# B&R Automation Studio project Parker_BMM_ST_V5_3147_V12 (part 2)

### Acp10map.ncm - 5PPC2100_BY01_000/Motion/Acp10map.ncm
```
NcMapping (NcSwId=Acp10, DisabledNodesAreHidden=True)
  NcObject 8V1090.001-2_ncV_AXIS1 (ModuleId=8V1090.001-2_L_BlowPin, Type=ncV_AXIS, Channel=1, Disabled=TRUE, ModuleDisabled=FALSE)
  NcObject 8V1090.001-2a_ncV_AXIS1 (ModuleId=8V1090.001-2a_R_BlowPin, Type=ncV_AXIS, Channel=1, Disabled=TRUE, ModuleDisabled=FALSE)
  NcObject 8V1180.001-2_ncV_AXIS1 (ModuleId=8V1180.001-2_L_Carriage, Type=ncV_AXIS, Channel=1, Disabled=TRUE, ModuleDisabled=FALSE)
  NcObject 8V1180.001-2a_ncV_AXIS1 (ModuleId=8V1180.001-2a_R_Carriage, Type=ncV_AXIS, Channel=1, Disabled=TRUE, ModuleDisabled=FALSE)
  NcObject 8B0P0440HW00.001-1_ncAXIS2 (ModuleId=8B0P0440HW00.001-1, Type=ncAXIS, Channel=2, AcoposSimulation=Off, Disabled=TRUE, ModuleDisabled=FALSE)
  NcObject 8B0P0440HW00.001-1_ncV_AXIS1 (ModuleId=8B0P0440HW00.001-1, Type=ncV_AXIS, Channel=1, Disabled=TRUE, ModuleDisabled=FALSE)
  NcObject 8B0P0440HW00.001-1_ncV_AXIS2 (ModuleId=8B0P0440HW00.001-1, Type=ncV_AXIS, Channel=2, Disabled=TRUE, ModuleDisabled=FALSE)
  NcObject 8BVI0110HWS0.000-1_ncAXIS2 (ModuleId=8BVI0110HWS0.000-1, Type=ncAXIS, Channel=2, AcoposSimulation=Off, Disabled=TRUE, ModuleDisabled=FALSE)
  NcObject 8BVI0110HWS0.000-1_ncV_AXIS1 (ModuleId=8BVI0110HWS0.000-1, Type=ncV_AXIS, Channel=1, Disabled=TRUE, ModuleDisabled=FALSE)
  NcObject 8BVI0110HWS0.000-1_ncV_AXIS2 (ModuleId=8BVI0110HWS0.000-1, Type=ncV_AXIS, Channel=2, Disabled=TRUE, ModuleDisabled=FALSE)
  NcObject gAxisBlowPinL (ModuleId=8V1090.001-2_L_BlowPin, Type=ncAXIS, Channel=1, AcoposSimulation=Off, InitParameter=BlowPinL, AcoposParameter=BlowPinLR, Disabled=TRUE, ModuleDisabled=FALSE)
  NcObject gAxisBlowPinR (ModuleId=8V1090.001-2a_R_BlowPin, Type=ncAXIS, Channel=1, AcoposSimulation=Off, InitParameter=BlowPinR, AcoposParameter=BlowPinLR, Disabled=TRUE, ModuleDisabled=FALSE)
  NcObject gAxisCarriageL (ModuleId=8V1180.001-2_L_Carriage, Type=ncAXIS, Channel=1, AcoposSimulation=Off, InitParameter=CarriageL, AcoposParameter=CarraigeLR, Disabled=TRUE, ModuleDisabled=FALSE)
  NcObject gAxisCarriageR (ModuleId=8V1180.001-2a_R_Carriage, Type=ncAXIS, Channel=1, AcoposSimulation=Off, InitParameter=CarriageR, AcoposParameter=CarraigeLR, Disabled=TRUE, ModuleDisabled=FALSE)
  NcObject 8BVI0330HWS0.000-1_ncAXIS2 (ModuleId=8BVI0330HWS0.000-1, Type=ncAXIS, Channel=2, AcoposSimulation=Off, Disabled=TRUE, ModuleDisabled=FALSE)
  NcObject 8BVI0330HWS0.000-1_ncV_AXIS1 (ModuleId=8BVI0330HWS0.000-1, Type=ncV_AXIS, Channel=1, Disabled=TRUE, ModuleDisabled=FALSE)
  NcObject 8BVI0330HWS0.000-1_ncV_AXIS2 (ModuleId=8BVI0330HWS0.000-1, Type=ncV_AXIS, Channel=2, Disabled=TRUE, ModuleDisabled=FALSE)
  NcObject 8BVI0330HWS0.000-1a_ncAXIS2 (ModuleId=8BVI0330HWS0.000-1a, Type=ncAXIS, Channel=2, AcoposSimulation=Off, Disabled=TRUE, ModuleDisabled=FALSE)
  NcObject 8BVI0330HWS0.000-1a_ncV_AXIS1 (ModuleId=8BVI0330HWS0.000-1a, Type=ncV_AXIS, Channel=1, Disabled=TRUE, ModuleDisabled=FALSE)
  NcObject 8BVI0330HWS0.000-1a_ncV_AXIS2 (ModuleId=8BVI0330HWS0.000-1a, Type=ncV_AXIS, Channel=2, Disabled=TRUE, ModuleDisabled=FALSE)
  NcObject 8BVI0110HWD0.000-1_ncV_AXIS1 (ModuleId=8BVI0110HWD0.000-1, Type=ncV_AXIS, Channel=1, Disabled=TRUE, ModuleDisabled=FALSE)
  NcObject 8BVI0110HWD0.000-1_ncV_AXIS2 (ModuleId=8BVI0110HWD0.000-1, Type=ncV_AXIS, Channel=2, Disabled=TRUE, ModuleDisabled=FALSE)
  NcObject 8BVI0440HWS0.000-1a_ncAXIS2 (ModuleId=8BVI0440HWS0.000-1a, Type=ncAXIS, Channel=2, AcoposSimulation=Off, Disabled=TRUE, ModuleDisabled=FALSE)
  NcObject 8BVI0440HWS0.000-1a_ncV_AXIS1 (ModuleId=8BVI0440HWS0.000-1a, Type=ncV_AXIS, Channel=1, Disabled=TRUE, ModuleDisabled=FALSE)
  NcObject 8BVI0440HWS0.000-1a_ncV_AXIS2 (ModuleId=8BVI0440HWS0.000-1a, Type=ncV_AXIS, Channel=2, Disabled=TRUE, ModuleDisabled=FALSE)
  NcObject 8BVI0028HWD0.000-1_ncV_AXIS1 (ModuleId=8BVI0028HWD0.000-1, Type=ncV_AXIS, Channel=1, Disabled=TRUE, ModuleDisabled=FALSE)
  NcObject 8BVI0028HWD0.000-1_ncV_AXIS2 (ModuleId=8BVI0028HWD0.000-1, Type=ncV_AXIS, Channel=2, Disabled=TRUE, ModuleDisabled=FALSE)
  NcObject gAxisTransferR (ModuleId=8BVI0110HWS0.000-1, Type=ncAXIS, Channel=1, AcoposSimulation=Off, InitParameter=TransferR, AcoposParameter=Tansfer, Disabled=TRUE, ModuleDisabled=FALSE)
  NcObject gAxisTransferR (ModuleId=8BVI0110HWS0.000-1, Type=ncAXIS, Channel=1, AcoposSimulation=Off, InitParameter=TransferR, AcoposParameter=Tansfer, Disabled=TRUE, ModuleDisabled=FALSE)
  NcObject gAxisCarriageL (ModuleId=8BVI0330HWS0.000-1a, Type=ncAXIS, Channel=1, AcoposSimulation=Off, InitParameter=CarriageL, AcoposParameter=CarraigeLR, Disabled=TRUE, ModuleDisabled=FALSE)
  NcObject 8BVI0330HWS0.000-1b_ncAXIS2 (ModuleId=8BVI0330HWS0.000-1b, Type=ncAXIS, Channel=2, AcoposSimulation=Off, Disabled=TRUE, ModuleDisabled=FALSE)
  NcObject 8BVI0330HWS0.000-1b_ncV_AXIS1 (ModuleId=8BVI0330HWS0.000-1b, Type=ncV_AXIS, Channel=1, Disabled=TRUE, ModuleDisabled=FALSE)
  NcObject 8BVI0330HWS0.000-1b_ncV_AXIS2 (ModuleId=8BVI0330HWS0.000-1b, Type=ncV_AXIS, Channel=2, Disabled=TRUE, ModuleDisabled=FALSE)
  NcObject 8BVI0440HWS0.000-1_ncAXIS2 (ModuleId=8BVI0440HWS0.000-1, Type=ncAXIS, Channel=2, AcoposSimulation=Off, Disabled=TRUE, ModuleDisabled=FALSE)
  NcObject 8BVI0440HWS0.000-1_ncV_AXIS1 (ModuleId=8BVI0440HWS0.000-1, Type=ncV_AXIS, Channel=1, Disabled=TRUE, ModuleDisabled=FALSE)
  NcObject 8BVI0440HWS0.000-1_ncV_AXIS2 (ModuleId=8BVI0440HWS0.000-1, Type=ncV_AXIS, Channel=2, Disabled=TRUE, ModuleDisabled=FALSE)
  NcObject gAxisClampR (ModuleId=8BVI0440HWS0.000-1, Type=ncAXIS, Channel=1, AcoposSimulation=Off, InitParameter=ClampR, AcoposParameter=ClampLR, Disabled=FALSE, ModuleDisabled=FALSE)
  NcObject gAxisClampR (ModuleId=8BVI0330HWS0.000-1b, Type=ncAXIS, Channel=1, AcoposSimulation=Off, InitParameter=ClampR, AcoposParameter=ClampLR, Disabled=TRUE, ModuleDisabled=FALSE)
  NcObject gAxisClampL (ModuleId=8BVI0440HWS0.000-1a, Type=ncAXIS, Channel=1, AcoposSimulation=Off, InitParameter=ClampL, AcoposParameter=ClampLR, Disabled=TRUE, ModuleDisabled=FALSE)
  NcObject gAxisExtrlift (ModuleId=8BVI0028HWD0.000-1, Type=ncAXIS, Channel=1, AcoposSimulation=Off, InitParameter=ExtrLift1, AcoposParameter=ExtrLift2, Disabled=FALSE, ModuleDisabled=FALSE)
  NcObject gAxisTransferR (ModuleId=8BVI0028HWD0.000-1, Type=ncAXIS, Channel=2, AcoposSimulation=Off, InitParameter=TransferR, AcoposParameter=Tansfer, Disabled=FALSE, ModuleDisabled=FALSE)
  NcObject gAxisPwr (ModuleId=8B0P0440HW00.001-1, Type=ncAXIS, Channel=1, AcoposSimulation=Off, InitParameter=Power, AcoposParameter=Power1, Disabled=FALSE, ModuleDisabled=FALSE)
  NcObject gAxisCarriageR (ModuleId=8BVI0330HWS0.000-1, Type=ncAXIS, Channel=1, AcoposSimulation=Off, InitParameter=CarriageR, AcoposParameter=CarraigeLR, Disabled=FALSE, ModuleDisabled=FALSE)
  NcObject gAxisThick (ModuleId=8BVI0110HWD0.000-1, Type=ncAXIS, Channel=1, AcoposSimulation=Off, InitParameter=ThickInit, AcoposParameter=ThickPara, Disabled=FALSE, ModuleDisabled=FALSE)
  NcObject gAxisBlowPinR (ModuleId=8BVI0110HWD0.000-1, Type=ncAXIS, Channel=2, AcoposSimulation=Off, InitParameter=BlowPinR, AcoposParameter=BlowPinLR, Disabled=FALSE, ModuleDisabled=FALSE)
```

## Configuration AR000

CPU PC_any, AutomationRuntime D4.26, Build 4.1.2, Vc V4.26.8, Safety 0.0

### Task classes (Cpu.sw)
```
Cyclic#1 (cycle 2000 us, tolerance 0 us):
  tk1_in <- In_Out.tk1_in.prg
  timer <- process.timer.prg
  length <- process.length.prg
  clamp <- process.clamp.prg
  carriage <- process.carriage.prg
  blowpin <- process.blowpin.prg
  tk1_out <- In_Out.tk1_out.prg
Cyclic#2 (cycle 10000 us, tolerance 100000 us):
  h_pwm <- Heating.h_pwm.prg
  tk2_io <- In_Out.tk2_io.prg
Cyclic#3 (cycle 4000 us, tolerance 100000 us):
  extrlift <- process.extrlift.prg
  cutter <- process.cutter.prg
  cutneck <- process.cutneck.prg
  cooldef <- process.cooldef.prg
  blowdef <- process.blowdef.prg
  bdeflash <- process.bdeflash.prg
  tdeflash <- process.tdeflash.prg
  inerpin <- process.inerpin.prg
  highblow <- process.highblow.prg
  lowblow <- process.lowblow.prg
  coolpin <- process.coolpin.prg
  coolpin2 <- process.coolpin2.prg
  coolpin3 <- process.coolpin3.prg
  submold <- process.submold.prg
  pinpart <- process.pinpart.prg
  screw <- process.screw.prg
  sealer <- process.sealer.prg
  bblowpin <- process.bblowpin.prg
  support <- process.support.prg
  tonnage <- process.tonnage.prg
  robot <- process.robot.prg
  extruder <- machine.extruder.prg
  extru_plk <- machine.extru_plk.prg
  autorun <- process.autorun.prg
Cyclic#4 (cycle 20000 us, tolerance 200000 us):
  keyled <- screen.keyled.prg
  manual <- machine.manual.prg
  calib <- machine.calib.prg
  reset <- machine.reset.prg
  workmode <- machine.workmode.prg
  mode <- machine.mode.prg
  panel <- screen.panel.prg
  hmi_cpy <- screen.hmi_cpy.prg
  pump <- machine.pump.prg
  mac_lubr <- machine.mac_lubr.prg
  oil_accu <- machine.oil_accu.prg
  mbusMaster <- comm.mbusMaster.prg
Cyclic#5 (cycle 500000 us, tolerance 500000 us):
  h_pid <- Heating.h_pid.prg
Cyclic#8 (cycle 200000 us, tolerance 30000000 us):
  spc_ctrl <- spc.spc_ctrl.prg
  trend <- Heating.trend.prg
  h_plan <- Heating.h_plan.prg
  scrshot <- screen.scrshot.prg
  hmiset <- screen.hmiset.prg
  password <- screen.password.prg
  modem <- comm.modem.prg
  vpn <- screen.vpn.prg
  recipe <- recipeMan.recipe.prg
  multsave <- recipeMan.multsave.prg
  oncesave <- recipeMan.oncesave.prg
  cfg_cpy <- recipeMan.cfg_cpy.prg
  pvchg <- VarChgLog.pvchg.prg
  alarm <- machine.alarm.prg
  epl <- comm.epl.prg
  energy <- machine.energy.prg
DataObjects: mb_cmd <- comm.mb_cmd.dob, pv_chg <- VarChgLog.pv_chg.dob, var_fix <- recipeMan.var_fix.dob, var_mold <- recipeMan.var_mold.dob, cfg_dat <- recipeMan.cfg_dat.dob, Acp10sys
VcDataObjects: visu15 <- Visu.visu15.dob
Binaries: TCData, visu1502, vccnum, vcpdvnc, vccalarm, vccovl, vcshared, vcfile, vccstr, vccline, arial, vcctrend, vcchtml, vcgclass, tahomabd, vccbtn, vcrt, vccdbox, visu1503, vcclbox, simsun, vcctext, vccbmp, vcfntttf, vcalarm, vcdsint, vcnet, visu1501, vccshape, vcchspot, arialbd, vctcal, vcmgr, vcdsloc, myxh, visvc, tahoma, vccurl, vccdt, vccbar, vcpfar00, vcpdsw, vcxml, vccscale, vcbclass, iomap, sysconf, ashwd, asfw, User, arconfig, Role, Acp10map, acp10cfg
Libraries: visapi, FileIO, runtime, sys_lib, standard, operator, dvframe, DataObj, Convert, brsystem, astime, asstring, AsIO, AsArLog, AsARCfg, Motorky, DRV_mbus, LoopConR, SimpFun, HydCtrl, NcGlobal, Acp10par, Acp10_MC, AsEPL, powerlnk, vcresman, ashydcon
```

### Hardware
```
PC : PC_any v1.1.0.0 (OrderNumber=PC)
  Connector IF3:
    Vnc1
    VncVcObjectName1 = visu15
    VncAuthentication1 = 1
    VncPasswordViewOnly1 = 1
    VncPasswordViewControl1 = 2
  ConfigurationID = bmm_AR000
  PermanentPvSize = 10000
  RemanentGlobalPvSize = 20000
  SystemTick = 2000
  TaskClassIdleTime = 2000
  Cyclic1Duration = 2000
  Cyclic1Tolerance = 0
  Cyclic1Output = 1
  Cyclic2Duration = 10000
  Cyclic2Tolerance = 100000
  Cyclic3Duration = 4000
  Cyclic3Tolerance = 100000
  Cyclic4Duration = 20000
  Cyclic4Tolerance = 200000
  Cyclic5Duration = 500000
  Cyclic5Tolerance = 500000
  Cyclic5Stack = 20000
  Cyclic6Duration = 30000
  Cyclic6Tolerance = 3000000
  Cyclic7Duration = 90000
  Cyclic7Tolerance = 9000000
  Cyclic8Duration = 200000
  Cyclic8Tolerance = 30000000
  Cyclic8Stack = 30000
```

### Acp10cfg.ncc - PC/Motion/Acp10cfg.ncc
```
NcConfiguration (Version=2.52.5, NcSwId=Acp10)
  ACP10CF1_typ:
    cnt_nettrc_rec_drive = 150
    bufsize_trace_upload = 1200
    tc_nc_man_task = Cyclic #1
    glob_pv_as_ncobject = Yes
    ncsys_dl_broadcast = Yes
    ncsys_dl_acp_reset = Yes
    safemc_log_err_to_ax = Yes
    network_init:
      ncsw_init_execute = Yes
      automatic_execute = No
      node_nr_warning = Yes
      net_err_before_ncact = Yes
    nettrc:
      enter_parsecrec = Yes
      enter_ncaction = Yes
      save_ring_startidx = No
    cam_prof_download:
      cam_dat_dl_parallel = No
      tc_cam_dl_parallel = Task class for NC Manager task
```

## Logical view

Binary libraries used (declarations not repeated): visapi, FileIO, runtime, sys_lib, standard, operator, dvframe, DataObj, Convert, brsystem, astime, asstring, AsIO, AsArLog, AsARCfg, Motorky 2.16.0, DRV_mbus, LoopConR 2.80.2, vcscrsht 4.24.0, HydCtrl 1.03.0, AsHydCon 3.10.0, AsEPL, Acp10man 5.06.1, Acp10par 5.06.1, NcGlobal 5.06.1, Acp10sim 5.06.1, Acp10_MC 5.06.1

### Package Logical/GlobalIncludes - Global include file

### draw.h
```c
#ifndef draw_h_
#define draw_h_

#define VSCREEN_WIDTH               302
#define VSCREEN_HEIGHT              402
#define VSCREEN_X0_POSITION         150
#define VSCREEN_Y0_POSITION          85

#define VSCREEN_COLOR_WEIGHT        169
#define VSCREEN_COLOR_BACKGROUND    140
#define VSCREEN_COLOR_FOCUS_LINE  	 51
#define VSCREEN_COLOR_UNFOCUS_LINE 	200
#define VSCREEN_COLOR_CURVE  	       46

#define VSCREEN_COLOR_CROSS_CURSOR 	 44
#define VSCREEN_COLOR_FRAME      	  0

#define S$THICK_POINT		   400
#define S$THICK_X_LENGTH		3000

#define S$THICK_INIT_LENGTH   300

#define S$THICK_SAMPLE		   100
#define S$THICK_MAX		      399
#define S$THICK_V_SCALE		   4

#define S$STEP_EDIT			10
#define S$STEP_ADDLINE     20
#define S$STEP_DELLINE	   30
#define S$STEP_CURVETOL		40
#define S$STEP_CURVEMOVE	50
#define S$STEP_UNDO			60
#define S$STEP_REDO			65
#define S$STEP_CLAER			70

#endif
```

### keyap880.h
```c
#ifndef keyap880_h_
#define keyap880_h_

#define S$KEYMATRIX_MAXCOUNT    400

#define OFFSET_EX2_01            216

/*  0 -- 39 AP880 key */
#define S$KEYMATRIX_MAIN_PUMP   	   0
#define S$KEYMATRIX_PARISON_PUMP 	1
#define S$KEYMATRIX_EXTRUDER_A   	2
#define S$KEYMATRIX_EXTRUDER_B   	3

#define S$KEYMATRIX_MODE_CALIB   	4
#define S$KEYMATRIX_MODE_MANUAL  	5
#define S$KEYMATRIX_MODE_AUTO    	6
#define S$KEYMATRIX_AUTO_RESET   	7
#define S$KEYMATRIX_CUTTER_FW   		8
#define S$KEYMATRIX_EXTRUDER_UP  	9
#define S$KEYMATRIX_LUBRICATION     10
#define S$KEYMATRIX_ALARM_RESET     11

#define S$KEYMATRIX_F1   				12
#define S$KEYMATRIX_F2   				13
#define S$KEYMATRIX_F3   				14
#define S$KEYMATRIX_F4   				15
#define S$KEYMATRIX_F5   				16
#define S$KEYMATRIX_F6   				17
#define S$KEYMATRIX_F7   				18
#define S$KEYMATRIX_F8   				19
#define S$KEYMATRIX_F9   				20
#define S$KEYMATRIX_F10   				21
#define S$KEYMATRIX_F11   				22
#define S$KEYMATRIX_F12   				23
#define S$KEYMATRIX_F13   				24
#define S$KEYMATRIX_F14   				25
#define S$KEYMATRIX_F15   				26
#define S$KEYMATRIX_F16   				27

#define S$KEYMATRIX_CARRIAGE_UP  	28
#define S$KEYMATRIX_CARRIAGE_DN  	29
#define S$KEYMATRIX_CLAMP_OPN   		30
#define S$KEYMATRIX_CLAMP_CLS   		31
#define S$KEYMATRIX_BLOWPIN_UP   	32
#define S$KEYMATRIX_BLOWPIN_DN   	33
#define S$KEYMATRIX_TOP_DEFLASH_FW  34
#define S$KEYMATRIX_BOT_DEFLASH_FW  35
#define S$KEYMATRIX_ROBOT_FW   		36
#define S$KEYMATRIX_ROBOT_BW   		37
#define S$KEYMATRIX_ROBOT_DN   		38
#define S$KEYMATRIX_ROBOT_CLS 		39

/*   5AC800EXT2-01 key   offset 216 */
#define S$KEYMATRIX_NUM7   		 	60
#define S$KEYMATRIX_NUM8   		 	61
#define S$KEYMATRIX_NUM9   		 	62
#define S$KEYMATRIX_NUM4   		 	64
#define S$KEYMATRIX_NUM5   		 	65
#define S$KEYMATRIX_NUM6   		 	66
#define S$KEYMATRIX_NUM1   		 	68
#define S$KEYMATRIX_NUM2   			69
#define S$KEYMATRIX_NUM3   		 	70
#define S$KEYMATRIX_NUM0   		 	73

#define S$KEYMATRIX_ESC    		 	63
#define S$KEYMATRIX_DEL			 		67
#define S$KEYMATRIX_ENTER  	     	71
#define S$KEYMATRIX_TAB          	77
#define S$KEYMATRIX_UP					75
#define S$KEYMATRIX_DOWN				79
#define S$KEYMATRIX_LEFT				76
#define S$KEYMATRIX_RIGHT				78

/* reserve key  */
#define S$KEYMATRIX_TOP_DEFLASH_BW  101
#define S$KEYMATRIX_ROBOT_UP   		102

#define S$KEYMATRIX_ROBOT_REJECT    103
#define S$KEYMATRIX_ROBOT_RESET 		104
#define S$KEYMATRIX_SUPPORT   		105
#define S$KEYMATRIX_SPEED_UP   		106
#define S$KEYMATRIX_SPEED_DN   	   107
#define S$KEYMATRIX_COOL_DEFLASH    108
#define S$KEYMATRIX_BLOW         	109
#define S$KEYMATRIX_BLOW_LOW        110
#define S$KEYMATRIX_COOL_DN         111
#define S$KEYMATRIX_COOL_BLOW			112
#define S$KEYMATRIX_SERVO_VALVE   	113
#define S$KEYMATRIX_AUTO_LUB   		114
#define S$KEYMATRIX_DIEGAP_UP      	115
#define S$KEYMATRIX_DIEGAP_DN  	   116
#define S$KEYMATRIX_FEED_OPEN       117
#define S$KEYMATRIX_VISU_EXTRUDER   118
#define S$KEYMATRIX_CUT_NECK  	   119

#define S$KEYMATRIX_PLATE_UP        120
#define S$KEYMATRIX_PLATE_DN        121
#define S$KEYMATRIX_SUBMOLD_OPN	   122
#define S$KEYMATRIX_SUBMOLD_CLS		123
#define S$KEYMATRIX_PIN_PART_FW  	124
#define S$KEYMATRIX_PIN_PART_BW	   125
#define S$KEYMATRIX_HANDLE_PUNCHER  126
#define S$KEYMATRIX_SCREW_FW	      131
#define S$KEYMATRIX_SCREW_BW  	   132
#define S$KEYMATRIX_COOL1_DN  	   133
#define S$KEYMATRIX_COOL1_BLOW  	   134
#define S$KEYMATRIX_COOL2_DN	      135
#define S$KEYMATRIX_COOL3_DN		   136
#define S$KEYMATRIX_VACCUM  	      137
//#define S$KEYMATRIX_HEAT_POWER      138
#define S$KEYMATRIX_MINOR_PUMP      139
#define S$KEYMATRIX_PENU_VALVE      140
#define S$KEYMATRIX_COOLING_PUMP   	141
#define S$KEYMATRIX_SENSOR_UP       142
#define S$KEYMATRIX_SENSOR_DN       143
#define S$KEYMATRIX_SENSOR_BOTTLE   144
#define S$KEYMATRIX_HOPPER_A   	   145
#define S$KEYMATRIX_DRY_CYCLE    	147

#endif
```

### pic_id.h
```c
#ifndef __pic_id_H__
#define __pic_id_H__

#define	PIC_INIT		          0

#define  PIC_OVERVIEW          	1

#define  PIC_TEMP_SET_1			4
#define  PIC_TEMP_SET_2   		5
#define  PIC_TEMP_EXTRUDER_2     6
#define  PIC_TEMP_EXTRUDER_3     7
#define  PIC_TEMP_EXTRUDER_4     8

#define  PIC_TEMP_DIEHEAD_1      9
#define  PIC_TEMP_DIEHEAD_2      10
#define  PIC_TEMP_DIEHEAD_3      11
#define  PIC_TEMP_DIEHEAD_4      12

#define  PIC_HEATING_PLAN        13
#define	PIC_TEMP_CONSTRUCT	   	14
#define	PIC_TEMP_CONSTRUCT_2	15

#define	PIC_TEMP_TRACE_1		16
#define	PIC_TEMP_TRACE_2		17
#define	PIC_TEMP_TRACE_3		18
#define	PIC_TEMP_TRACE_4		19
#define	PIC_TEMP_TRACE_5		20
#define	PIC_TEMP_TRACE_6		21
#define	PIC_TEMP_TRACE_7		22
#define	PIC_TEMP_TRACE_8		23

#define	PIC_TEMP_OPT_1		   24
#define	PIC_TEMP_OPT_2		   25
#define	PIC_TEMP_OPT_3		   26
#define	PIC_TEMP_OPT_4		   27
#define	PIC_TEMP_OPT_5		   28
#define	PIC_TEMP_OPT_6		   29
#define	PIC_TEMP_OPT_7		   30
#define	PIC_TEMP_OPT_8		   31

#define	PIC_TEMP_CONFIG_1		32
#define	PIC_TEMP_CONFIG_2		33
#define	PIC_TEMP_CONFIG_3		34
#define	PIC_TEMP_CONFIG_4		35
#define	PIC_TEMP_CONFIG_5		36
#define	PIC_TEMP_CONFIG_6		37
#define	PIC_TEMP_CONFIG_7		38
#define	PIC_TEMP_CONFIG_8		39

#define  PIC_TIME_1           41
#define  PIC_TIME_2          	42
#define  PIC_TIME_3          	43
#define  PIC_TIME_4          	44
#define  PIC_TIME_5          	45
#define  PIC_TIME_6          	46
#define  PIC_TIME_7          	47
#define  PIC_TIME_8          	48
#define  PIC_TIME_9          	49

#define  PIC_CLAMP_L            51
#define  PIC_CLAMP_R            52
#define  PIC_TRANSPORT_L        53
#define  PIC_TRANSPORT_R        54
#define  PIC_ROBOT_L			55
#define  PIC_ROBOT_R			56

#define  PIC_DEFLASH			58
#define  PIC_BOTTOM_DEFLASH       60
#define  PIC_BLOW_PIN_L      	  61
#define  PIC_BLOW_PIN_R      	  62
#define  PIC_BLOW_PIN2_L      	  1061
#define  PIC_BLOW_PIN2_R      	  1062
#define  PIC_BLOW_PIN_CONFIG    63
#define  PIC_SUBMOLD            64
#define  PIC_EXTRLIFT           65

#define  PIC_ACCU_SETTING       68
#define  PIC_CALIB_SETTING       69
#define  PIC_CALIB_SETTING_2     70

#define  PIC_OPTION             71
#define  PIC_RECIPE			    72
#define  PIC_OPTION_2           73

#define  PIC_SPEED			     75
#define  PIC_LENGTH			     76

#define PIC_THICK_START			81
#define	PIC_CURVE_EDIT			82
#define	PIC_CURVE_TRACE			83
#define	PIC_MARKER_SET_A		86
#define PIC_CURVEDATA_A			87
#define	PIC_MARKER_SET_B		88
#define PIC_CURVEDATA_B        	89
#define	PIC_IO_DO_2  			90
#define	PIC_IO_DI_1  			91
#define	PIC_IO_DI_2  			92
#define	PIC_IO_DI_3  			93
#define	PIC_IO_DO_1  			94
#define	PIC_IO_DO_3  			95
#define	PIC_IO_DO_4  			96
#define	PIC_IO_AI_1  			97
#define	PIC_IO_AO_1  			98
#define	PIC_IO_MODULE  			99
#define	PIC_IO_DRIVER_1    		100
#define	PIC_IO_DRIVER_2    		101
#define	PIC_ENERGY_MONITOR_ALL  102
#define	PIC_ENERGY_MONITOR   	103

#define PIC_AUTO_STEP			104
#define PIC_AUTO_START			105
#define	PIC_SPC_CTRL			106
#define	PIC_SPC_1				107
#define	PIC_SPC_2				108

#define	PIC_ALARM_CURRENT	   	111
#define	PIC_ALARM_HISTORY		112
#define	PIC_ALARM_1				113
#define	PIC_ALARM_2				114
#define	PIC_ALARM_3				115
#define	PIC_ALARM_4				116
#define	PIC_ALARM_5				117

#define	PIC_PASSWORD_LOGIN      120
#define	PIC_SYSTEM_SET_1		121
#define	PIC_SYSTEM_SET_2		122
#define	PIC_SYSTEM_SET_3		123

#define	PIC_INDUSTY_40			  	125

#define	PIC_PASSWORD_SET			130
#define	PIC_PROPORTION_VALVE		133
//#define	PIC_VALVE_DELAY	    	134
#define	PIC_PRESSURE_CALIBRATION   	134
#define	PIC_IP_CONFIG		    	135
#define	PIC_PV_LOG		        	136
#define	PIC_LOG_INFO		    	137
#define	PIC_VNC						138
#define	PIC_HIGH_PASSWORD       	139

#define	PIC_INIT_SET				140
#define PIC_GAP_CALIBRATE			141
#define	PIC_ACCU_CALIBRATE			142
#define	PIC_DEFAULT_SET				143
#define	PIC_GAP_CALIBRATE_HELP  	145
#define	PIC_THICK_DIVER  			146

#define	PIC_SCREEN_CALIBRATE	150
#define	PIC_MOTOR_TREND  		151

#define PIC_FAST_SETTING		160

#define  PIC_CONFIG_HELP        170
#define  PIC_CLAMP_CONFIG       171
#define  PIC_TRANSPORT_CONFIG   172
#define  PIC_BLOW_PIN_CONFIG    173
#define  PIC_EXTRLIFT_CONFIG   	174

#define	PIC_OEM_SETTING_1		180
#define	PIC_OEM_SETTING_2		181
#define	PIC_OEM_SETTING_3		182
#define	PIC_OEM_SETTING_4		183

#define	PIC_OEM_SETTING_10		189

#define  PIC_CLAMP_TOGGLE       190
#define  PIC_CARRIAGE_TOGGLE    191
#define  PIC_EXTRLIFT_TOGGLE    192

#define	PIC_SCREEN_SAVE			200

#define	PIC_CALIB_CLAMP_ENCODER		220
#define	PIC_CALIB_CARRIAGE_ENCODER	221
#define	PIC_CALIB_BLOWPIN_ENCODER	222
#define	PIC_CALIB_OTHER_ENCODER		223
#define	PIC_CALIB_ROBOT_ENCODER		224
#define	PIC_CALIB_CLAMP_LVDT		226
#define	PIC_CALIB_CARRIAGE_LVDT		227
#define	PIC_CALIB_BLOWPIN_LVDT		228
#define	PIC_CALIB_OTHER_LVDT		229

#endif
```

### recipe.h
```c
#ifndef receipe_h_
#define receipe_h_

#define S$NUM_RECIPE    50

#endif/* #ifndef receipe_h_ */
```

### defines.h
```c
#ifndef __DEFINES_H__
#define __DEFINES_H__

#define MODE_NOTHING              10
#define MODE_MANUAL               20
#define MODE_AUTO                 30
#define MODE_SEMI_AUTO            35
#define MODE_ADJUST               40

/* ------------------------------------------------------------------- */
#define  CONTROL_STAT_ACTIVE    1
/* ------------------------------------------------------------------- */

#define  S$STATUS_AUTORUN           1
#define  S$STATUS_CALIBRATE         2
#define  S$STATUS_MANUAL            3
#define  S$STATUS_NEED_CALIBRATE    4

#define  ABS(X)   (((X) > 0.0) ? (X) : (-1.0*(X)))

#endif /* #ifndef __DEFINES_H__ */
```

### thick.h
```c
#ifndef _THICK_H_
#define _THICK_H_

#define 	STEP_THICK_READY    	     0
#define 	STEP_THICK_AUTO_RUN     100
#define 	STEP_THICK_CALIB_UP   	5000
#define 	STEP_THICK_CALIB_DOWN 	15000
#define  STEP_THICK_STOP         20000

#define	THICK_NUM				   100
/*number of thickness points            壁厚控制点数*/
#define  TIME_OF_CYCLE             2
/*cyclic time of timer1                 高速任务循环时间*/
#define  NOFOCUS                   0
#define	THICK_RANGE					300

/************** thickness control function ********************/
void TimeCurveData(Thick_Data_typ *);
void AccuCurveData(Thick_Data_typ *);
void PIDCtrl(Thick_PID_typ * pPID);
int  ISqrt(long n);                             /* 整型开平方 */
/****************************************************/
#endif /* _THICK_H_ end */
```

### edge.h
```c
/***************************************************************************************/
/*		 Include for Edge Detection											  		               */
/*-------------------------------------------------------------------------------------*/
/*		 Filename:	   edge.h												  		                  */
/*       Author:       B&R				                                      		         */
/*       Date:         24.07.2001                                             		   */
/***************************************************************************************/
/* Description:                                                            	  		   */
/*	Macros for Edgedetection. This macros uses a special feature of the GNU compiler:   */
/*	"Statements and Declarations in Expressions" see more details in GNU-Documentation  */
/*	So they may not work with other compilers.										            */
/*																					                        */
/*	EDGEPOS  Detection of positive transition of signal  							            */
/*	EDGENEG  Detection of negative transition of signal 							            */
/*	EDGE     Detection of positive and negative transition of signal 				         */
/*                                                                            		   */
/***************************************************************************************/

#ifndef __EDGE_H__
#define __EDGE_H__

/*****************************************************************************************/
/*	EDGEPOS  return 1 at positive transition of signal, in all other cases 0 is returned */
/*****************************************************************************************/
#define EDGEPOS(variable,__buffer)	\
({plcbit result; 					      \
	if (variable && !__buffer)       \
    {								         \
       	result=1;                  \
    }								         \
    else                            \
    {								         \
       	result=0;                  \
    }								         \
    __buffer=variable;              \
    result;                         \
})

/*****************************************************************************************/
/*	EDGENEG  return 1 at negative transition of signal, in all other cases 0 is returned */
/*****************************************************************************************/
#define EDGENEG(variable,__buffer) 	\
({plcbit result; 					      \
	if (!variable && __buffer)       \
    {								         \
       	result=1;                  \
    }								         \
    else                            \
    {								         \
       	result=0;                  \
    }								         \
    __buffer=variable;              \
    result;                         \
})

/**************************************************************************************************/
/*	EDGE return 1 at positive and negative transition of signal, in all other cases 0 is returned */
/**************************************************************************************************/
#define EDGE(variable,__buffer)		\
({plcbit result; 					      \
	if (variable != __buffer)        \
    {								         \
       	result=1;                  \
    }								         \
    else                            \
    {								         \
       	result=0;                  \
    }								         \
    __buffer=variable;              \
    result;                         \
})

#endif /*__EDGE_H__*/
```

### keyap2100.h
```c
#ifndef keyapPPC2100_1505_h_
#define keyapPPC2100_1505_h_

#define S$KEYMATRIX_MAXCOUNT    400

#define OFFSET_EX2_01            216

/*  0 -- 9 PPC2100  Left Key */
#define S$KEYMATRIX_CUTTER_FW		0
#define S$KEYMATRIX_EXTRUDER_UP		1
#define S$KEYMATRIX_CARRIAGE_UP		2
#define S$KEYMATRIX_CARRIAGE_DN		3
#define S$KEYMATRIX_CLAMP_CLS		4
#define S$KEYMATRIX_CLAMP_OPN		5
#define S$KEYMATRIX_BLOWPIN_DN		6
#define S$KEYMATRIX_BLOWPIN_UP		7
#define S$KEYMATRIX_BLOW			8
#define S$KEYMATRIX_HOOK_PIN_FW 	9
/* 10 -- 21 PPC2100 Middle Key */

#define S$KEYMATRIX_TOP_DEFLASH_FW	10
#define S$KEYMATRIX_TOP_DEFLASH_BW	11
#define S$KEYMATRIX_ROBOT_FW		12
#define S$KEYMATRIX_ROBOT_CLS		13
#define S$KEYMATRIX_COOL_DN			14
#define S$KEYMATRIX_COOL_BLOW		15
#define S$KEYMATRIX_COOL2_DN		16
#define S$KEYMATRIX_COOL2_BLOW		17
#define S$KEYMATRIX_COOL3_DN		18
#define S$KEYMATRIX_COOL3_BLOW		19
#define S$KEYMATRIX_SUBMOLD_OPN		20
#define S$KEYMATRIX_SUBMOLD_CLS		21

//#define S$KEYMATRIX_BLOW			12
//#define S$KEYMATRIX_PRODUCTAUX_CLS	13
//#define S$KEYMATRIX_ROBOT_FWBW		14
//#define S$KEYMATRIX_ROBOT_CLS		15

/* 22 -- 31 PPC2100 Right Key */

#define S$KEYMATRIX_HEAT_POWER		22
//#define S$KEYMATRIX_EXTRUDER_A_PLK	23
//#define S$KEYMATRIX_EXTRUDER_B_PLK	24
//#define S$KEYMATRIX_EXTRUDER_C_PLK	25

/*for ABB inveter ------------------------------*/
#define S$KEYMATRIX_EXTRUDER_A_ABB	23
#define S$KEYMATRIX_EXTRUDER_D_ABB	24
#define S$KEYMATRIX_EXTRUDER_B_ABB	25
#define S$KEYMATRIX_EXTRUDER_C_ABB	26
#define S$KEYMATRIX_EXTRUDER_V_ABB	153 //Follow Extruder_D
/*-----------------------------------------------*/
//#define S$KEYMATRIX_EXTRUDER_V_ABB	26

#define S$KEYMATRIX_PARISON_PUMP	100

#define S$KEYMATRIX_MAIN_PUMP		27
#define S$KEYMATRIX_MODE_MANUAL		28
#define S$KEYMATRIX_MODE_AUTO		29
#define S$KEYMATRIX_AUTO_STOP		30
#define S$KEYMATRIX_MODE_CALIB		31

/*200 -- 215 Visual Funcion Key*/

#define S$KEYMATRIX_F1   				200
#define S$KEYMATRIX_F2   				201
#define S$KEYMATRIX_F3   				202
#define S$KEYMATRIX_F4   				203
#define S$KEYMATRIX_F5   				204
#define S$KEYMATRIX_F6   				205
#define S$KEYMATRIX_F7   				206
#define S$KEYMATRIX_F8   				207
#define S$KEYMATRIX_F9   				208
#define S$KEYMATRIX_F10   				209
#define S$KEYMATRIX_F11   				210
#define S$KEYMATRIX_F12   				211
#define S$KEYMATRIX_F13   				212
#define S$KEYMATRIX_F14   				213
#define S$KEYMATRIX_F15   				214
#define S$KEYMATRIX_F16   				215

/*Auto Reset*/

#define S$KEYMATRIX_AUTO_RESET			100

/* reserve key  */

#define S$KEYMATRIX_NUM7   		 	60
#define S$KEYMATRIX_NUM8   		 	61
#define S$KEYMATRIX_NUM9   		 	62
#define S$KEYMATRIX_NUM4   		 	64
#define S$KEYMATRIX_NUM5   		 	65
#define S$KEYMATRIX_NUM6   		 	66
#define S$KEYMATRIX_NUM1   		 	68
#define S$KEYMATRIX_NUM2   			69
#define S$KEYMATRIX_NUM3   		 	70
#define S$KEYMATRIX_NUM0   		 	73

#define S$KEYMATRIX_ESC    		 	63
#define S$KEYMATRIX_DEL			 	67
#define S$KEYMATRIX_ENTER  	     	71
#define S$KEYMATRIX_TAB          	77
#define S$KEYMATRIX_UP				75
#define S$KEYMATRIX_DOWN			79
#define S$KEYMATRIX_LEFT			76
#define S$KEYMATRIX_RIGHT			78

//#define S$KEYMATRIX_TOP_DEFLASH_BW  101
//#define S$KEYMATRIX_ROBOT_FW   		102
#define S$KEYMATRIX_ROBOT_BW   		103
#define S$KEYMATRIX_ROBOT_OPN    	104
//#define S$KEYMATRIX_ROBOT_CLS 		105
#define S$KEYMATRIX_SUPPORT   		106
#define S$KEYMATRIX_SPEED_UP   		107
#define S$KEYMATRIX_SPEED_DN   	    108
#define S$KEYMATRIX_COOL_DEFLASH    109
#define S$KEYMATRIX_BLOW_LOW        110

#define S$KEYMATRIX_SERVO_VALVE   	113
#define S$KEYMATRIX_AUTO_LUB   		114
#define S$KEYMATRIX_DIEGAP_UP      	115
#define S$KEYMATRIX_DIEGAP_DN  	    116
#define S$KEYMATRIX_FEED_OPEN       117
//#define S$KEYMATRIX_VISU_EXTRUDER	118
#define S$KEYMATRIX_CUT_NECK		119

//#define S$KEYMATRIX_COOL_DN		111
//#define S$KEYMATRIX_COOL_BLOW		112
//#define S$KEYMATRIX_COOL2_DN		133
//#define S$KEYMATRIX_COOL2_BLOW	134
//#define S$KEYMATRIX_COOL3_DN		120
//#define S$KEYMATRIX_COOL3_BLOW	121
#define S$PAGE_FAST_SEETING			122

#define S$KEYMATRIX_PULL_BOTTOM_FW  123
#define S$KEYMATRIX_PIN_PART_FW  	124
#define S$KEYMATRIX_PIN_PART_BW	   	125
#define S$KEYMATRIX_HANDLE_PUNCHER  126
//#define S$KEYMATRIX_HOOK_PIN_FW   127
//#define S$KEYMATRIX_EXTRUDER_UP	128
#define S$KEYMATRIX_EXTRUDER_DN		129
#define S$KEYMATRIX_SCREW_FW	    131
#define S$KEYMATRIX_SCREW_BW  	    132
#define S$PAGE_FAST_SEETING 		134
#define S$KEYMATRIX_BLOWPINDN_HOLD	135
#define S$KEYMATRIX_BOTSUBMOLD_OPN	136
#define S$KEYMATRIX_VACCUM  	    137
#define S$KEYMATRIX_BOTSUBMOLD_CLS  138
#define S$KEYMATRIX_MINOR_PUMP      139
#define S$KEYMATRIX_PENU_VALVE      140
#define S$KEYMATRIX_COOLING_PUMP   	141
#define S$KEYMATRIX_SENSOR_UP       142
#define S$KEYMATRIX_SENSOR_DN       143
#define S$KEYMATRIX_SENSOR_BOTTLE   144
#define S$KEYMATRIX_HOPPER_A   	    145
#define S$KEYMATRIX_DRY_CYCLE    	147

#define S$KEYMATRIX_BOT_DEFLASH_FW   	148
#define S$KEYMATRIX_BOT_DEFLASH_BW   	149
//#define S$KEYMATRIX_SUBMOLD_OPN   	150
//#define S$KEYMATRIX_SUBMOLD_CLS 		151

#define S$KEYMATRIX_LUBRICATION     152

#define S$KEYMATRIX_EXTRUDER_A		154
#define S$KEYMATRIX_EXTRUDER_B		155
#define S$KEYMATRIX_EXTRUDER_C		156
#define S$KEYMATRIX_VISU_EXTRUDER	157
#define S$KEYMATRIX_VISU_EXTRUDER_PLK	158
#define S$KEYMATRIX_ALARM_RESET		159
//#define S$PAGE_FAST_SEETING			160

#define S$KEYMATRIX_PLATE_UP		161
#define S$KEYMATRIX_PLATE_DN		162
#define S$KEYMATRIX_PLATE_FW		163
#define S$KEYMATRIX_PLATE_BW		164

#endif
```

### Sizing.var - size of recipe array and task
```iecst
(********************************************************************
 * COPYRIGHT --  B&R
 ********************************************************************
 * File: Sizing.var
 * Author: lij
 * Created: December 19, 2013
 ********************************************************************
 * Global Sizing var of project BMM
 ********************************************************************)
(*Key and object Max*)
VAR CONSTANT
	MAX_KEY_COUNT : UINT := 400;
	MAX_OBJECT : USINT := 100;
END_VAR
(*Trend curve number*)
VAR CONSTANT
	TREND_CURVE_NUM : USINT := 40;
END_VAR
(*temperature idex and group ---> MAX*)
VAR CONSTANT
	MAX_IDX_ZONE : USINT := 40; (*Max. Heating zone index  ---- recipe*)
	MAX_IDX_CONTRL_ZONES : USINT := 33; (*Max. Control Heating zone index*)
	MAX_IDX_TEMPGROUP : USINT := 2; (*Max. Heating group index   ----- recipe*)
END_VAR
(*third axis control ---> MAX*)
VAR CONSTANT
	MAX_AXIS_NUM : USINT := 2; (*Max Axis number*)
END_VAR
(*Alarm index and text ---> MAX*)
VAR CONSTANT
	MAX_ALARM_NUM : UINT := 500; (*Max alarm number*)
	MAX_ALARM_TEXT : UINT := 120; (*Max alarm text length*)
END_VAR
(*Log information buffer length*)
VAR CONSTANT
	MAX_LOG_BUFFER : USINT := 27; (*Max log buffer length*)
END_VAR
(*Frequency inventor*)
VAR CONSTANT
	MAX_IDX_COMM : USINT := 3;
	MAX_IDX_CONROL_COMM : USINT := 2;
END_VAR
(*Energy Monitor Module*)
VAR CONSTANT
	MAX_IDX_ENERGY : USINT := 3;
	MAX_TOGGLE_LIN_NUM : USINT := 30;
END_VAR
```

### Enums.typ
```iecst
(*Axes Configuration*)

TYPE
	actuator_typ_enum :
		( (*Axes Actuator types *)
		ACTUATOR_UNDEFINED := 0, (* Actuator: undefined *)
		ACTUATOR_HYD := 1, (* Actuator: Hydraulic *)
		ACTUATOR_PNEU := 2, (* Actuator: Pneumatic *)
		ACTUATOR_ELECTRIC := 3 (* Actuator: Electric drive *)
		);
END_TYPE

(*Electric*)

TYPE
	mechanism_typ_enum :
		(
		MECHANISM_LINEAR := 0,
		MECHANISM_TOGGLE := 1
		);
END_TYPE

(*Hydraulic*)

TYPE
	valve_typ_enum :
		(
		VALVE_UNDEFINED := 0,
		VALVE_DIR := 1,
		VALVE_PROP := 2
		);
	sensor_type_enum :
		(
		SENSOR_UNDEFINED := 0,
		SENSOR_LVDT := 1,
		SENSOR_SWITCH := 2
		);
	pressure_output_enum :
		(
		PRESSURE_OUTPUT_UNDEFINED := 0,
		PRESSURE_OUTPUT_SYSTEM_SINGLE := 1,
		PRESSURE_OUTPUT_ACC := 2,
		PRESSURE_OUTPUT_ACC_EXTRLIFT := 3,
		PRESSURE_OUTPUT_NONE := 4
		);
	flux_output_enum :
		(
		FLUX_OUTPUT_UNDEFINED := 0,
		FLUX_OUTPUT_SYSTEM_SINGLE := 1,
		FLUX_OUTPUT_PROP_VALVE_SINGLE := 2,
		FLUX_OUTPUT_ACC := 3,
		FLUX_OUTPUT_ACC_EXTRLIFT := 4,
		FLUX_OUTPUT_NONE := 5
		);
END_TYPE

(*Extruder*)

TYPE
	extruder_ctrl_typ_enum :
		(
		CTRL_UNDEFINED := 0,
		CTRL_VF := 1,
		CTRL_ABB_POWERLINK := 2
		);
END_TYPE

(*Blow*)

TYPE
	blow_mode_enum :
		(
		BLOW_MODE_STANDARD := 0,
		BLOW_MODE_FREEZINGBLOW := 1,
		New_Member1,
		New_Member
		);
END_TYPE

(*Support Air*)

TYPE
	supportair_mode_enum :
		(
		SUPPORTAIR_MODE_STANDARD := 0,
		SUPPORTAIR_MODE_AFTER_CLAMP_CLS := 1,
		New_Member3,
		New_Member2
		);
END_TYPE
```
